TYPE typ_MotionHoming :
STRUCT
	MC_Home						: MC_Home;
END_STRUCT
END_TYPE

(* stored: Version 1.1.0.1, ProductVersion 3.1.4022.17
   DUT typ_MotionHoming: Id {2b05828a-303b-4515-b241-5f15c7436456} *)
